(* CoDeSys 2.3 export: TYPE_LED_RGB_CONFIG.EXP *)

(* Data type *)
TYPE Type_LED_RGB_CONFIG :
STRUCT
	Speed_RANDOM	:REAL;

	tDimmTime: 		REAL	:= 5000;
	bDimmOnMode:	BOOL	:= TRUE;
	tDimmOnTime:		REAL	:= 500;
	bDimmOffMode:	BOOL	:= TRUE;
	tDimmOffTime:		REAL	:= 1000;
END_STRUCT
END_TYPE
